(*
SPDX-FileCopyrightText: © 2026 Oleksandr Tiutyk <trofimich@gmail.com>
SPDX-License-Identifier: MIT
License: https://opensource.org/license/mit
*)

{attribute 'no_explicit_call' := 'do not call this function block directly'} 
PROGRAM SignedInt16
VAR CONSTANT
	MIN_VALUE : INT := -32_768;
	MAX_VALUE : INT := +32_767;
END_VAR
VAR
	{attribute 'hide'} 
	_ClassName : STRING := __POUNAME();
END_VAR

{attribute 'monitoring' := 'call'}
PROPERTY ClassName : REFERENCE TO STRING
GET
ClassName REF= _ClassName;
END_GET
END_PROPERTY

{attribute 'monitoring' := 'call'}
PROPERTY NamespaceName : REFERENCE TO STRING
GET
NamespaceName REF= CurrentNamespace.Name;
END_GET
END_PROPERTY

END_PROGRAM

(* stored: Version 1.1.0.1
   POU SignedInt16: Id {68b7f7f9-8120-432b-9159-ae2909b3c9a5}, SpecialFunc None
   Property ClassName: Id {ec30b879-6a8e-4528-a927-021b411518a1}
   Get Get: Id {7c84c451-d33c-4e35-b9fc-78ccb1ef882d}
   Property NamespaceName: Id {5834a303-0ddd-45d7-9348-42eb8fe1576e}
   Get Get: Id {c07abbc7-e3b7-4197-932c-29282e11d83a} *)
